// TIA Portal V17 export
// export: Created 2025-03-07T09:18:47.277747Z, ExportSetting WithDefaults, DisplayName Totally Integrated Automation Portal, DisplayVersion V17 Update 8, DisplayName TIA Portal Openness, DisplayVersion V17 Update 8, DisplayName TIA Portal Version Control Interface, DisplayVersion V17, DisplayName SINAMICS Startdrive Advanced, DisplayVersion V17 SP2, DisplayName SINAMICS Startdrive G110M, G120, G120C, G120D, G120P, G115D, DisplayVersion V17 SP2, DisplayName SINAMICS Startdrive G130, G150, S120, S150, SINAMICS MV, S210, DisplayVersion V17 SP2, DisplayName STEP 7 Professional, DisplayVersion V17 Update 8, DisplayName SINUMERIK ONE STEP 7 Toolbox, DisplayVersion V17 Update 12, DisplayName SINUMERIK 840D sl STEP 7 Toolbox, DisplayVersion V17 Update 12, DisplayName STEP 7 Safety, DisplayVersion V17 Update 6, DisplayName WinCC Advanced, DisplayVersion V17 Update 8
FUNCTION_BLOCK "FB6501_MEAS_DEVICE_HATCH"   // FB6501, LAD
{ S7_Optimized_Access := 'FALSE' }
AUTHOR : ETXETAR
VERSION : 1.0
// stored: AutoNumber false, IsIECCheckEnabled false, SetENOAutomatically false, UDAEnableTagReadback false
   VAR_INPUT
      OPTIONS_0 : Byte := 2#0000_0000;   // OPTIONS 0
      CLOSED_1_I : Bool;   // CLOSED 1 INPUT
      CLOSED_2_I : Bool;   // CLOSED 2 INPUT
      CLOSED_3_I : Bool;   // CLOSED 3 INPUT
      CLOSED_4_I : Bool;   // CLOSED 4 INPUT
      OPENED_1_I : Bool;   // OPEN 1 INPUT
      OPENED_2_I : Bool;   // OPEN 2 INPUT
      OPENED_3_I : Bool;   // OPEN 3 INPUT
      OPENED_4_I : Bool;   // OPEN 4 INPUT
      CLOSE_CONDITIONS : Bool;   // CLOSE CONDITIONS
      OPEN_CONDITIONS : Bool;   // OPEN CONDITIONS
      HMI_LINE_REQUEST : Bool;   // HMI LINE REQUEST
      CLOSE_AUTO_REQUEST : Bool;   // AUTO CLOSE REQUEST
      OPEN_AUTO_REQUEST_1 : Bool;   // AUTO OPEN REQUEST
      UNIT_ALARM : UInt;   // UNIT NUMBER MIN. NUMBER=1 MAX. NUMBER=4
      STATION_ALARM : UInt;   // STATION NUMBER MIN. NUMBER=0 MAX. NUMBER=4
   END_VAR
   VAR_OUTPUT
      CLOSED : Bool;   // CLOSED STATUS
      OPENED : Bool;   // OPENED STATUS
      CLOSED_1_ALARM : Bool;   // CLOSED 1 ALARM
      CLOSED_2_ALARM : Bool;   // CLOSED 2 ALARM
      CLOSED_3_ALARM : Bool;   // CLOSED 3 ALARM
      CLOSED_4_ALARM : Bool;   // CLOSED 4 ALARM
      OPENED_1_ALARM : Bool;   // OPENED 1 ALARM
      OPENED_2_ALARM : Bool;   // OPENED 2 ALARM
      OPENED_3_ALARM : Bool;   // OPENED 3 ALARM
      OPENED_4_ALARM : Bool;   // OPENED 4 ALARM
      HMI_MOTION_EXECUTABILITY_LEFT : Bool;   // HMI MOTION EXECUTABILITY LEFT
      HMI_MOTION_EXECUTABILITY_RIGHT : Bool;   // HMI MOTION EXECUTABILITY RIGHT
      HMI_MOTION_END_POS_LEFT : Bool;   // HMI MOTION END POSITION LEFT
      HMI_MOTION_END_POS_RIGHT : Bool;   // HMI MOTION END POSITION RIGHT
      HMI_MOTION_ACTIVE_LEFT : Bool;   // HMI MOTION ACTIVE LEFT
      HMI_MOTION_ACTIVE_RIGHT : Bool;   // HMI MOTION ACTIVE RIGHT
      CLOSE : Bool;   // CLOSE OUTPUT
      OPEN : Bool;   // OPEN OUTPUT
   END_VAR
   VAR DB_SPECIFIC
      CYL { S7_SetPoint := 'True'} : "OPEN_CLOSE_HATCH_CLADDING";
      TIMER_CLOSED { S7_SetPoint := 'True'} : TON_TIME;   // CLOSED TIMER
      TIMER_OPENED { S7_SetPoint := 'True'} : TON_TIME;   // OPENED TIMER
      TIMER_SIMULTANEITY { S7_SetPoint := 'True'} : TON_TIME;   // SIMULTANEITY TIMER
      TIMER_TIME_EXCEEDED { S7_SetPoint := 'True'} : TON_TIME;   // TIME EXCEEDED TIMER
   END_VAR
   VAR_TEMP
      INPUTS_MASK : Byte;   // INPUTS_MASK
      O_BYTE_0 : Struct   // OPTIONS BYTE 0
         CLOSED_INPUT_1 : Bool;   // CLOSED INPUT 1 OPTION
         CLOSED_INPUT_2 : Bool;   // CLOSED INPUT 2 OPTION
         CLOSED_INPUT_3 : Bool;   // CLOSED
         CLOSED_INPUT_4 : Bool;   // CLOSED INPUT 4 OPTION
         OPENED_INPUT_1 : Bool;   // OPENED INPUT 1 OPTION
         OPENED_INPUT_2 : Bool;   // OPENED INPUT 2 OPTION
         OPENED_INPUT_3 : Bool;   // OPENED INPUT 3 OPTION
         OPENED_INPUT_4 : Bool;   // OPENED INPUT 4 OPTION
      END_STRUCT;
      DB_NUMBER : DInt;   // DB NUMBER FOR ALARM AND HELP DECODING
   END_VAR
   // TIMER_CLOSED.PT := T#100MS;
   // TIMER_OPENED.PT := T#300MS;
   // TIMER_SIMULTANEITY.PT := T#100MS;
   // TIMER_TIME_EXCEEDED.PT := T#8S;
   VAR_TEMP   // added for the SCL form of the ladder/FBD networks
      _w1 : Bool;
      _w2 : Bool;
   END_VAR
BEGIN

NETWORK
TITLE = READ INSTANCE DB
      L     DINO;
      +     10#800000;
      T     #DB_NUMBER;


REGION Network 2: OPTIONS
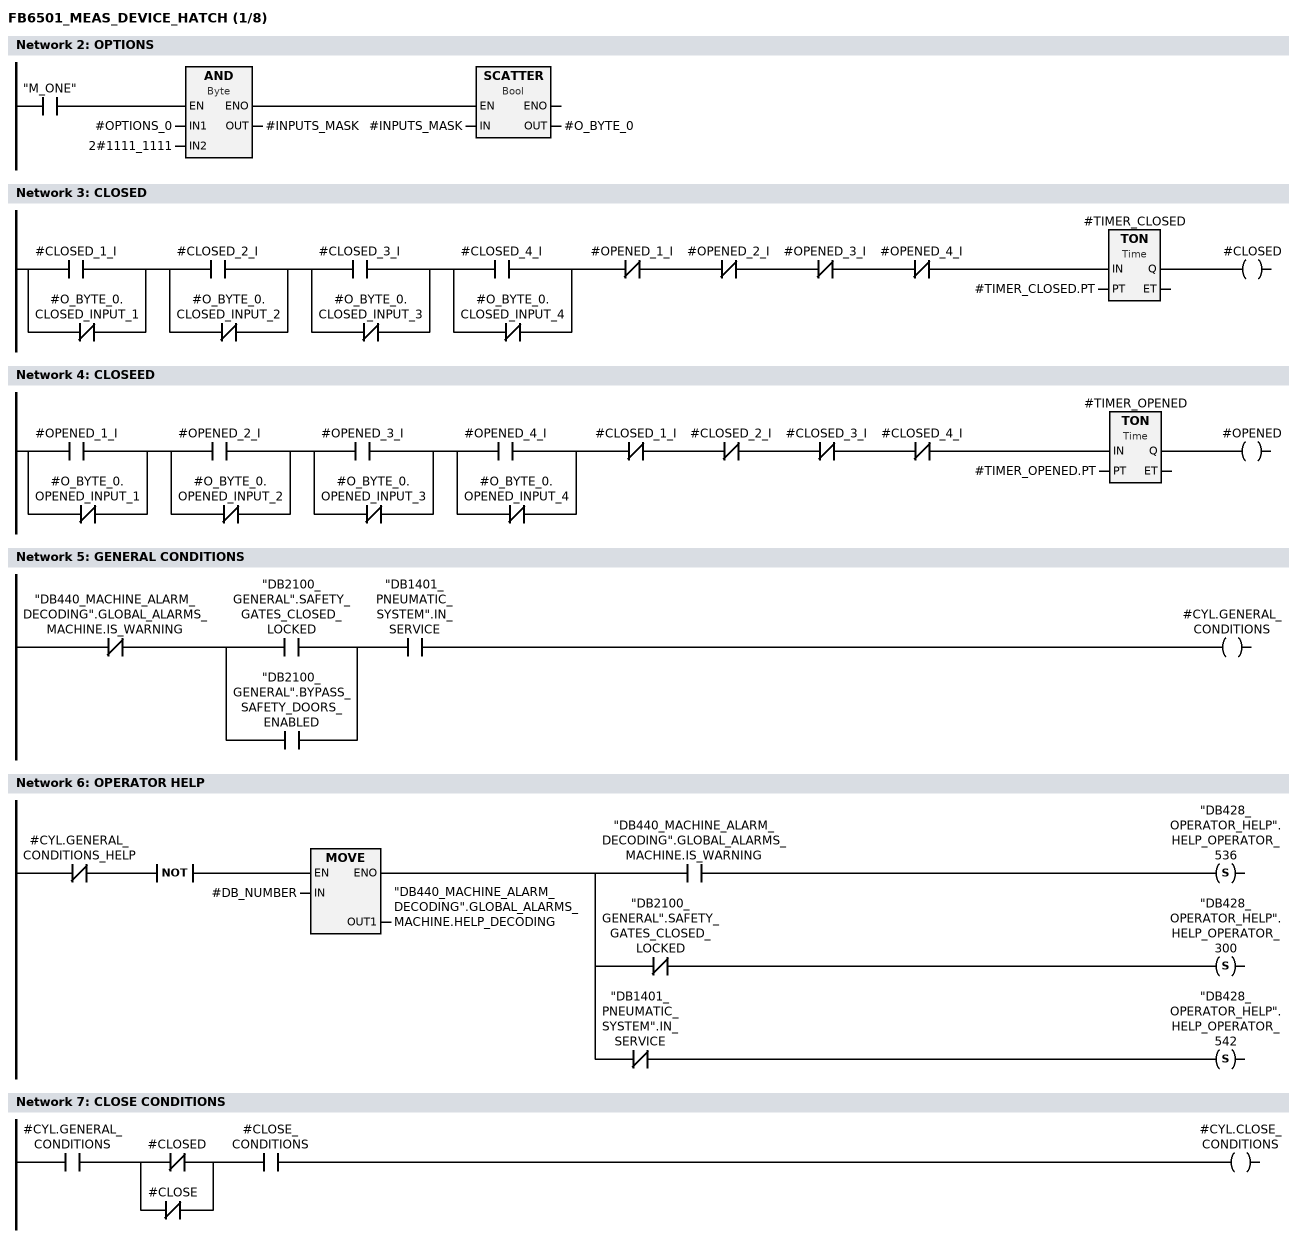
   RUNG wire#powerrail
      Contact( "M_ONE" )
      { S7_Templates := "SrcType := Byte"; S7_GenerateENO := "TRUE" } And(in1 := #OPTIONS_0, in2 := 2#1111_1111, out => #INPUTS_MASK)
      { S7_Templates := "[dest_type := Bool, src_type := Byte]" } SCATTER(IN := #INPUTS_MASK, OUT => #O_BYTE_0)
   END_RUNG
   // the same network as SCL:
   IF "M_ONE" THEN
       #INPUTS_MASK := #OPTIONS_0 AND 2#1111_1111;
       SCATTER(IN := #INPUTS_MASK, OUT => #O_BYTE_0);
   END_IF;
END_REGION

REGION Network 3: CLOSED
   RUNG wire#powerrail
      Contact( #CLOSED_1_I )
      wire#w1
      Contact( #CLOSED_2_I )
      wire#w2
      Contact( #CLOSED_3_I )
      wire#w3
      Contact( #CLOSED_4_I )
      wire#w4
      I_Contact( #OPENED_1_I )
      I_Contact( #OPENED_2_I )
      I_Contact( #OPENED_3_I )
      I_Contact( #OPENED_4_I )
      { S7_Templates := "time_type := Time" } #TIMER_CLOSED.TON(pt := #TIMER_CLOSED.PT, et =>)
      Coil( #CLOSED )
   END_RUNG
   RUNG wire#powerrail
      I_Contact( #O_BYTE_0.CLOSED_INPUT_1 )
   END_RUNG wire#w1
   RUNG wire#w1
      I_Contact( #O_BYTE_0.CLOSED_INPUT_2 )
   END_RUNG wire#w2
   RUNG wire#w2
      I_Contact( #O_BYTE_0.CLOSED_INPUT_3 )
   END_RUNG wire#w3
   RUNG wire#w3
      I_Contact( #O_BYTE_0.CLOSED_INPUT_4 )
   END_RUNG wire#w4
   // the same network as SCL:
   #TIMER_CLOSED(IN := (#CLOSED_1_I OR NOT #O_BYTE_0.CLOSED_INPUT_1) AND (#CLOSED_2_I OR NOT #O_BYTE_0.CLOSED_INPUT_2) AND (#CLOSED_3_I OR NOT #O_BYTE_0.CLOSED_INPUT_3) AND (#CLOSED_4_I OR NOT #O_BYTE_0.CLOSED_INPUT_4) AND NOT #OPENED_1_I AND NOT #OPENED_2_I AND NOT #OPENED_3_I AND NOT #OPENED_4_I,   // TON
                 PT := #TIMER_CLOSED.PT);
   #CLOSED := #TIMER_CLOSED.Q;
END_REGION

REGION Network 4: CLOSEED
   RUNG wire#powerrail
      Contact( #OPENED_1_I )
      wire#w1
      Contact( #OPENED_2_I )
      wire#w2
      Contact( #OPENED_3_I )
      wire#w3
      Contact( #OPENED_4_I )
      wire#w4
      I_Contact( #CLOSED_1_I )
      I_Contact( #CLOSED_2_I )
      I_Contact( #CLOSED_3_I )
      I_Contact( #CLOSED_4_I )
      { S7_Templates := "time_type := Time" } #TIMER_OPENED.TON(pt := #TIMER_OPENED.PT, et =>)
      Coil( #OPENED )
   END_RUNG
   RUNG wire#powerrail
      I_Contact( #O_BYTE_0.OPENED_INPUT_1 )
   END_RUNG wire#w1
   RUNG wire#w1
      I_Contact( #O_BYTE_0.OPENED_INPUT_2 )
   END_RUNG wire#w2
   RUNG wire#w2
      I_Contact( #O_BYTE_0.OPENED_INPUT_3 )
   END_RUNG wire#w3
   RUNG wire#w3
      I_Contact( #O_BYTE_0.OPENED_INPUT_4 )
   END_RUNG wire#w4
   // the same network as SCL:
   #TIMER_OPENED(IN := (#OPENED_1_I OR NOT #O_BYTE_0.OPENED_INPUT_1) AND (#OPENED_2_I OR NOT #O_BYTE_0.OPENED_INPUT_2) AND (#OPENED_3_I OR NOT #O_BYTE_0.OPENED_INPUT_3) AND (#OPENED_4_I OR NOT #O_BYTE_0.OPENED_INPUT_4) AND NOT #CLOSED_1_I AND NOT #CLOSED_2_I AND NOT #CLOSED_3_I AND NOT #CLOSED_4_I,   // TON
                 PT := #TIMER_OPENED.PT);
   #OPENED := #TIMER_OPENED.Q;
END_REGION

REGION Network 5: GENERAL CONDITIONS
   RUNG wire#powerrail
      I_Contact( "DB440_MACHINE_ALARM_DECODING".GLOBAL_ALARMS_MACHINE.IS_WARNING )
      wire#w1
      Contact( "DB2100_GENERAL".SAFETY_GATES_CLOSED_LOCKED )
      wire#w2
      Contact( "DB1401_PNEUMATIC_SYSTEM".IN_SERVICE )
      Coil( #CYL.GENERAL_CONDITIONS )
   END_RUNG
   RUNG wire#w1
      Contact( "DB2100_GENERAL".BYPASS_SAFETY_DOORS_ENABLED )
   END_RUNG wire#w2
   // the same network as SCL:
   #CYL.GENERAL_CONDITIONS := NOT "DB440_MACHINE_ALARM_DECODING".GLOBAL_ALARMS_MACHINE.IS_WARNING AND ("DB2100_GENERAL".SAFETY_GATES_CLOSED_LOCKED OR "DB2100_GENERAL".BYPASS_SAFETY_DOORS_ENABLED) AND "DB1401_PNEUMATIC_SYSTEM".IN_SERVICE;
END_REGION

REGION Network 6: OPERATOR HELP
   RUNG wire#powerrail
      I_Contact( #CYL.GENERAL_CONDITIONS_HELP )
      Not()
      { S7_GenerateENO := "TRUE" } Move(in := #DB_NUMBER, out1 => "DB440_MACHINE_ALARM_DECODING".GLOBAL_ALARMS_MACHINE.HELP_DECODING)
      wire#w1
      Contact( "DB440_MACHINE_ALARM_DECODING".GLOBAL_ALARMS_MACHINE.IS_WARNING )
      S_Coil( "DB428_OPERATOR_HELP".HELP_OPERATOR_536 )
   END_RUNG
   RUNG wire#w1
      I_Contact( "DB2100_GENERAL".SAFETY_GATES_CLOSED_LOCKED )
      S_Coil( "DB428_OPERATOR_HELP".HELP_OPERATOR_300 )
   END_RUNG
   RUNG wire#w1
      I_Contact( "DB1401_PNEUMATIC_SYSTEM".IN_SERVICE )
      S_Coil( "DB428_OPERATOR_HELP".HELP_OPERATOR_542 )
   END_RUNG
   // the same network as SCL:
   // ENO of a box is taken as its EN; it also drops when the box reports an error
   #_w1 := NOT (NOT #CYL.GENERAL_CONDITIONS_HELP);
   IF #_w1 THEN "DB440_MACHINE_ALARM_DECODING".GLOBAL_ALARMS_MACHINE.HELP_DECODING := #DB_NUMBER; END_IF;
   IF #_w1 AND "DB440_MACHINE_ALARM_DECODING".GLOBAL_ALARMS_MACHINE.IS_WARNING THEN
       "DB428_OPERATOR_HELP".HELP_OPERATOR_536 := TRUE;
   END_IF;
   IF #_w1 AND NOT "DB2100_GENERAL".SAFETY_GATES_CLOSED_LOCKED THEN
       "DB428_OPERATOR_HELP".HELP_OPERATOR_300 := TRUE;
   END_IF;
   IF #_w1 AND NOT "DB1401_PNEUMATIC_SYSTEM".IN_SERVICE THEN
       "DB428_OPERATOR_HELP".HELP_OPERATOR_542 := TRUE;
   END_IF;
END_REGION

REGION Network 7: CLOSE CONDITIONS
   RUNG wire#powerrail
      Contact( #CYL.GENERAL_CONDITIONS )
      wire#w1
      I_Contact( #CLOSED )
      wire#w2
      Contact( #CLOSE_CONDITIONS )
      Coil( #CYL.CLOSE_CONDITIONS )
   END_RUNG
   RUNG wire#w1
      I_Contact( #CLOSE )
   END_RUNG wire#w2
   // the same network as SCL:
   #CYL.CLOSE_CONDITIONS := #CYL.GENERAL_CONDITIONS AND (NOT #CLOSED OR NOT #CLOSE) AND #CLOSE_CONDITIONS;
END_REGION

REGION Network 8: OPERATOR HELP
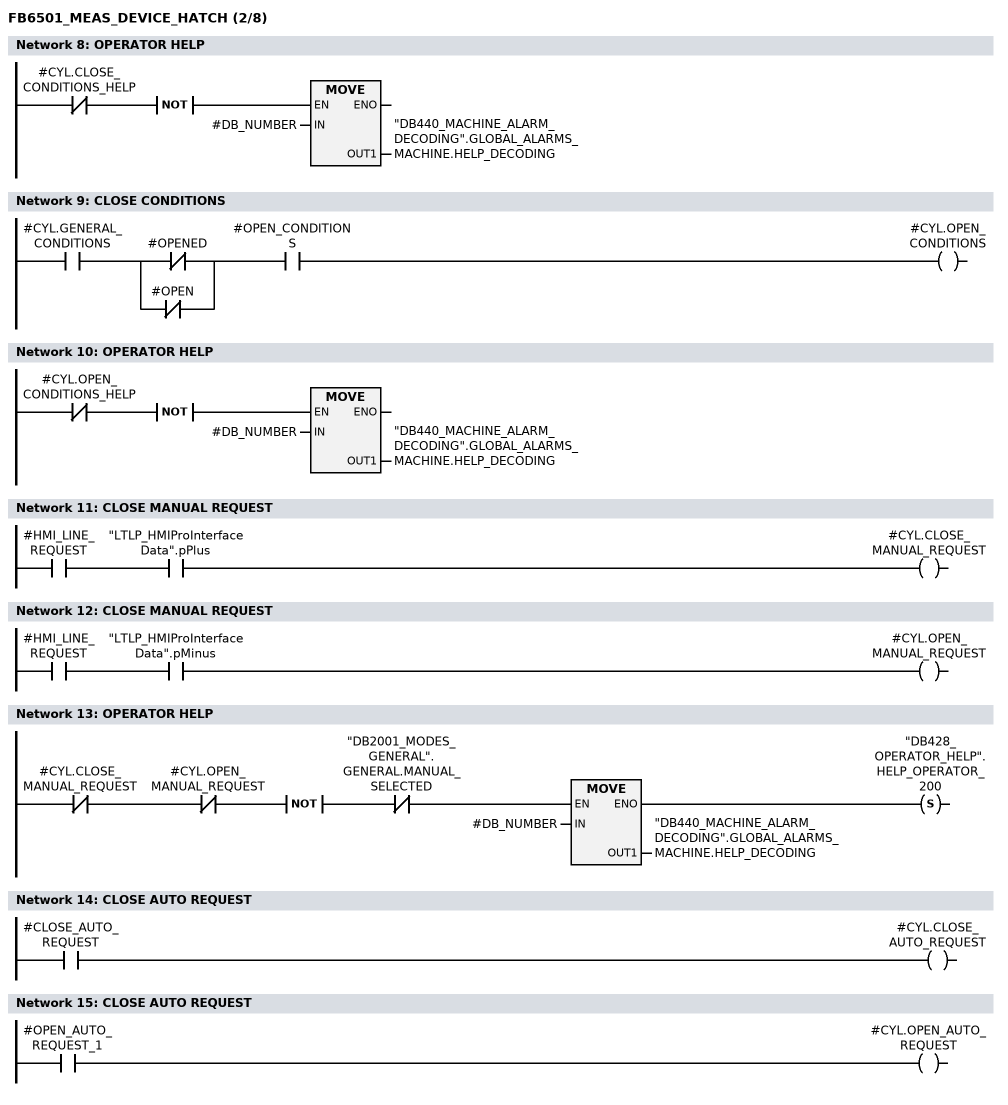
   RUNG wire#powerrail
      I_Contact( #CYL.CLOSE_CONDITIONS_HELP )
      Not()
      { S7_GenerateENO := "TRUE" } Move(in := #DB_NUMBER, out1 => "DB440_MACHINE_ALARM_DECODING".GLOBAL_ALARMS_MACHINE.HELP_DECODING)
   END_RUNG
   // the same network as SCL:
   IF NOT (NOT #CYL.CLOSE_CONDITIONS_HELP) THEN
       "DB440_MACHINE_ALARM_DECODING".GLOBAL_ALARMS_MACHINE.HELP_DECODING := #DB_NUMBER;
   END_IF;
END_REGION

REGION Network 9: CLOSE CONDITIONS
   RUNG wire#powerrail
      Contact( #CYL.GENERAL_CONDITIONS )
      wire#w1
      I_Contact( #OPENED )
      wire#w2
      Contact( #OPEN_CONDITIONS )
      Coil( #CYL.OPEN_CONDITIONS )
   END_RUNG
   RUNG wire#w1
      I_Contact( #OPEN )
   END_RUNG wire#w2
   // the same network as SCL:
   #CYL.OPEN_CONDITIONS := #CYL.GENERAL_CONDITIONS AND (NOT #OPENED OR NOT #OPEN) AND #OPEN_CONDITIONS;
END_REGION

REGION Network 10: OPERATOR HELP
   RUNG wire#powerrail
      I_Contact( #CYL.OPEN_CONDITIONS_HELP )
      Not()
      { S7_GenerateENO := "TRUE" } Move(in := #DB_NUMBER, out1 => "DB440_MACHINE_ALARM_DECODING".GLOBAL_ALARMS_MACHINE.HELP_DECODING)
   END_RUNG
   // the same network as SCL:
   IF NOT (NOT #CYL.OPEN_CONDITIONS_HELP) THEN
       "DB440_MACHINE_ALARM_DECODING".GLOBAL_ALARMS_MACHINE.HELP_DECODING := #DB_NUMBER;
   END_IF;
END_REGION

REGION Network 11: CLOSE MANUAL REQUEST
   RUNG wire#powerrail
      Contact( #HMI_LINE_REQUEST )
      Contact( "LTLP_HMIProInterfaceData".pPlus )
      Coil( #CYL.CLOSE_MANUAL_REQUEST )
   END_RUNG
   // the same network as SCL:
   #CYL.CLOSE_MANUAL_REQUEST := #HMI_LINE_REQUEST AND "LTLP_HMIProInterfaceData".pPlus;
END_REGION

REGION Network 12: CLOSE MANUAL REQUEST
   RUNG wire#powerrail
      Contact( #HMI_LINE_REQUEST )
      Contact( "LTLP_HMIProInterfaceData".pMinus )
      Coil( #CYL.OPEN_MANUAL_REQUEST )
   END_RUNG
   // the same network as SCL:
   #CYL.OPEN_MANUAL_REQUEST := #HMI_LINE_REQUEST AND "LTLP_HMIProInterfaceData".pMinus;
END_REGION

REGION Network 13: OPERATOR HELP
   RUNG wire#powerrail
      I_Contact( #CYL.CLOSE_MANUAL_REQUEST )
      I_Contact( #CYL.OPEN_MANUAL_REQUEST )
      Not()
      I_Contact( "DB2001_MODES_GENERAL".GENERAL.MANUAL_SELECTED )
      { S7_GenerateENO := "TRUE" } Move(in := #DB_NUMBER, out1 => "DB440_MACHINE_ALARM_DECODING".GLOBAL_ALARMS_MACHINE.HELP_DECODING)
      S_Coil( "DB428_OPERATOR_HELP".HELP_OPERATOR_200 )
   END_RUNG
   // the same network as SCL:
   // ENO of a box is taken as its EN; it also drops when the box reports an error
   IF NOT (NOT #CYL.CLOSE_MANUAL_REQUEST AND NOT #CYL.OPEN_MANUAL_REQUEST) AND NOT "DB2001_MODES_GENERAL".GENERAL.MANUAL_SELECTED THEN
       "DB440_MACHINE_ALARM_DECODING".GLOBAL_ALARMS_MACHINE.HELP_DECODING := #DB_NUMBER;
       "DB428_OPERATOR_HELP".HELP_OPERATOR_200 := TRUE;
   END_IF;
END_REGION

REGION Network 14: CLOSE AUTO REQUEST
   RUNG wire#powerrail
      Contact( #CLOSE_AUTO_REQUEST )
      Coil( #CYL.CLOSE_AUTO_REQUEST )
   END_RUNG
   // the same network as SCL:
   #CYL.CLOSE_AUTO_REQUEST := #CLOSE_AUTO_REQUEST;
END_REGION

REGION Network 15: CLOSE AUTO REQUEST
   RUNG wire#powerrail
      Contact( #OPEN_AUTO_REQUEST_1 )
      Coil( #CYL.OPEN_AUTO_REQUEST )
   END_RUNG
   // the same network as SCL:
   #CYL.OPEN_AUTO_REQUEST := #OPEN_AUTO_REQUEST_1;
END_REGION

REGION Network 16: CLOSE GLOBAL REQUEST
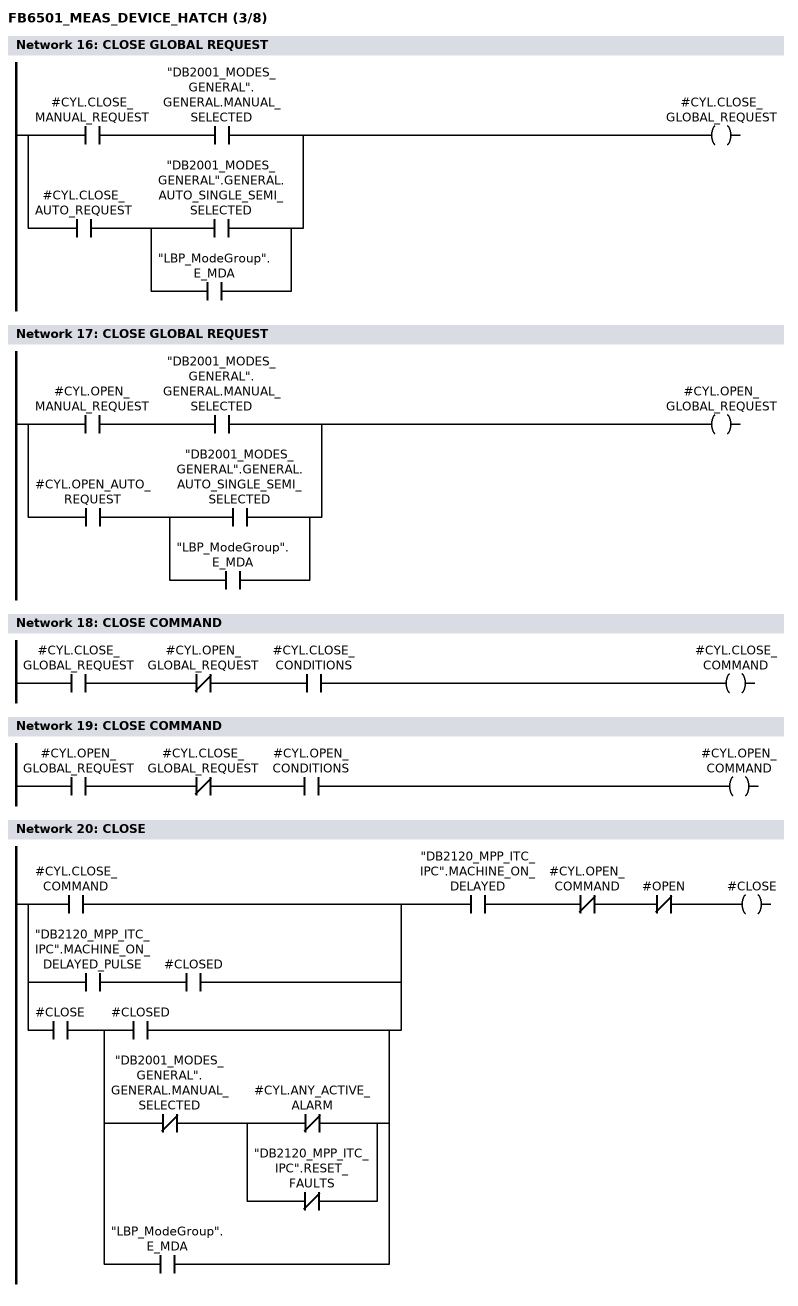
   RUNG wire#powerrail
      Contact( #CYL.CLOSE_MANUAL_REQUEST )
      Contact( "DB2001_MODES_GENERAL".GENERAL.MANUAL_SELECTED )
      wire#w1
      Coil( #CYL.CLOSE_GLOBAL_REQUEST )
   END_RUNG
   RUNG wire#powerrail
      Contact( #CYL.CLOSE_AUTO_REQUEST )
      wire#w2
      Contact( "DB2001_MODES_GENERAL".GENERAL.AUTO_SINGLE_SEMI_SELECTED )
   END_RUNG wire#w1
   RUNG wire#w2
      Contact( "LBP_ModeGroup".E_MDA )
   END_RUNG wire#w1
   // the same network as SCL:
   #CYL.CLOSE_GLOBAL_REQUEST := (#CYL.CLOSE_MANUAL_REQUEST AND "DB2001_MODES_GENERAL".GENERAL.MANUAL_SELECTED) OR (#CYL.CLOSE_AUTO_REQUEST AND ("DB2001_MODES_GENERAL".GENERAL.AUTO_SINGLE_SEMI_SELECTED OR "LBP_ModeGroup".E_MDA));
END_REGION

REGION Network 17: CLOSE GLOBAL REQUEST
   RUNG wire#powerrail
      Contact( #CYL.OPEN_MANUAL_REQUEST )
      Contact( "DB2001_MODES_GENERAL".GENERAL.MANUAL_SELECTED )
      wire#w1
      Coil( #CYL.OPEN_GLOBAL_REQUEST )
   END_RUNG
   RUNG wire#powerrail
      Contact( #CYL.OPEN_AUTO_REQUEST )
      wire#w2
      Contact( "DB2001_MODES_GENERAL".GENERAL.AUTO_SINGLE_SEMI_SELECTED )
   END_RUNG wire#w1
   RUNG wire#w2
      Contact( "LBP_ModeGroup".E_MDA )
   END_RUNG wire#w1
   // the same network as SCL:
   #CYL.OPEN_GLOBAL_REQUEST := (#CYL.OPEN_MANUAL_REQUEST AND "DB2001_MODES_GENERAL".GENERAL.MANUAL_SELECTED) OR (#CYL.OPEN_AUTO_REQUEST AND ("DB2001_MODES_GENERAL".GENERAL.AUTO_SINGLE_SEMI_SELECTED OR "LBP_ModeGroup".E_MDA));
END_REGION

REGION Network 18: CLOSE COMMAND
   RUNG wire#powerrail
      Contact( #CYL.CLOSE_GLOBAL_REQUEST )
      I_Contact( #CYL.OPEN_GLOBAL_REQUEST )
      Contact( #CYL.CLOSE_CONDITIONS )
      Coil( #CYL.CLOSE_COMMAND )
   END_RUNG
   // the same network as SCL:
   #CYL.CLOSE_COMMAND := #CYL.CLOSE_GLOBAL_REQUEST AND NOT #CYL.OPEN_GLOBAL_REQUEST AND #CYL.CLOSE_CONDITIONS;
END_REGION

REGION Network 19: CLOSE COMMAND
   RUNG wire#powerrail
      Contact( #CYL.OPEN_GLOBAL_REQUEST )
      I_Contact( #CYL.CLOSE_GLOBAL_REQUEST )
      Contact( #CYL.OPEN_CONDITIONS )
      Coil( #CYL.OPEN_COMMAND )
   END_RUNG
   // the same network as SCL:
   #CYL.OPEN_COMMAND := #CYL.OPEN_GLOBAL_REQUEST AND NOT #CYL.CLOSE_GLOBAL_REQUEST AND #CYL.OPEN_CONDITIONS;
END_REGION

REGION Network 20: CLOSE
   RUNG wire#powerrail
      Contact( #CYL.CLOSE_COMMAND )
      wire#w1
      Contact( "DB2120_MPP_ITC_IPC".MACHINE_ON_DELAYED )
      I_Contact( #CYL.OPEN_COMMAND )
      I_Contact( #OPEN )
      Coil( #CLOSE )
   END_RUNG
   RUNG wire#powerrail
      Contact( "DB2120_MPP_ITC_IPC".MACHINE_ON_DELAYED_PULSE )
      Contact( #CLOSED )
   END_RUNG wire#w1
   RUNG wire#powerrail
      Contact( #CLOSE )
      wire#w2
      Contact( #CLOSED )
   END_RUNG wire#w1
   RUNG wire#w2
      I_Contact( "DB2001_MODES_GENERAL".GENERAL.MANUAL_SELECTED )
      wire#w3
      I_Contact( #CYL.ANY_ACTIVE_ALARM )
   END_RUNG wire#w1
   RUNG wire#w3
      I_Contact( "DB2120_MPP_ITC_IPC".RESET_FAULTS )
   END_RUNG wire#w1
   RUNG wire#w2
      Contact( "LBP_ModeGroup".E_MDA )
   END_RUNG wire#w1
   // the same network as SCL:
   #CLOSE := (#CYL.CLOSE_COMMAND OR ("DB2120_MPP_ITC_IPC".MACHINE_ON_DELAYED_PULSE AND #CLOSED) OR (#CLOSE AND (#CLOSED OR (NOT "DB2001_MODES_GENERAL".GENERAL.MANUAL_SELECTED AND (NOT #CYL.ANY_ACTIVE_ALARM OR NOT "DB2120_MPP_ITC_IPC".RESET_FAULTS)) OR "LBP_ModeGroup".E_MDA))) AND "DB2120_MPP_ITC_IPC".MACHINE_ON_DELAYED AND NOT #CYL.OPEN_COMMAND AND NOT #OPEN;
END_REGION

REGION Network 21: CLOSE
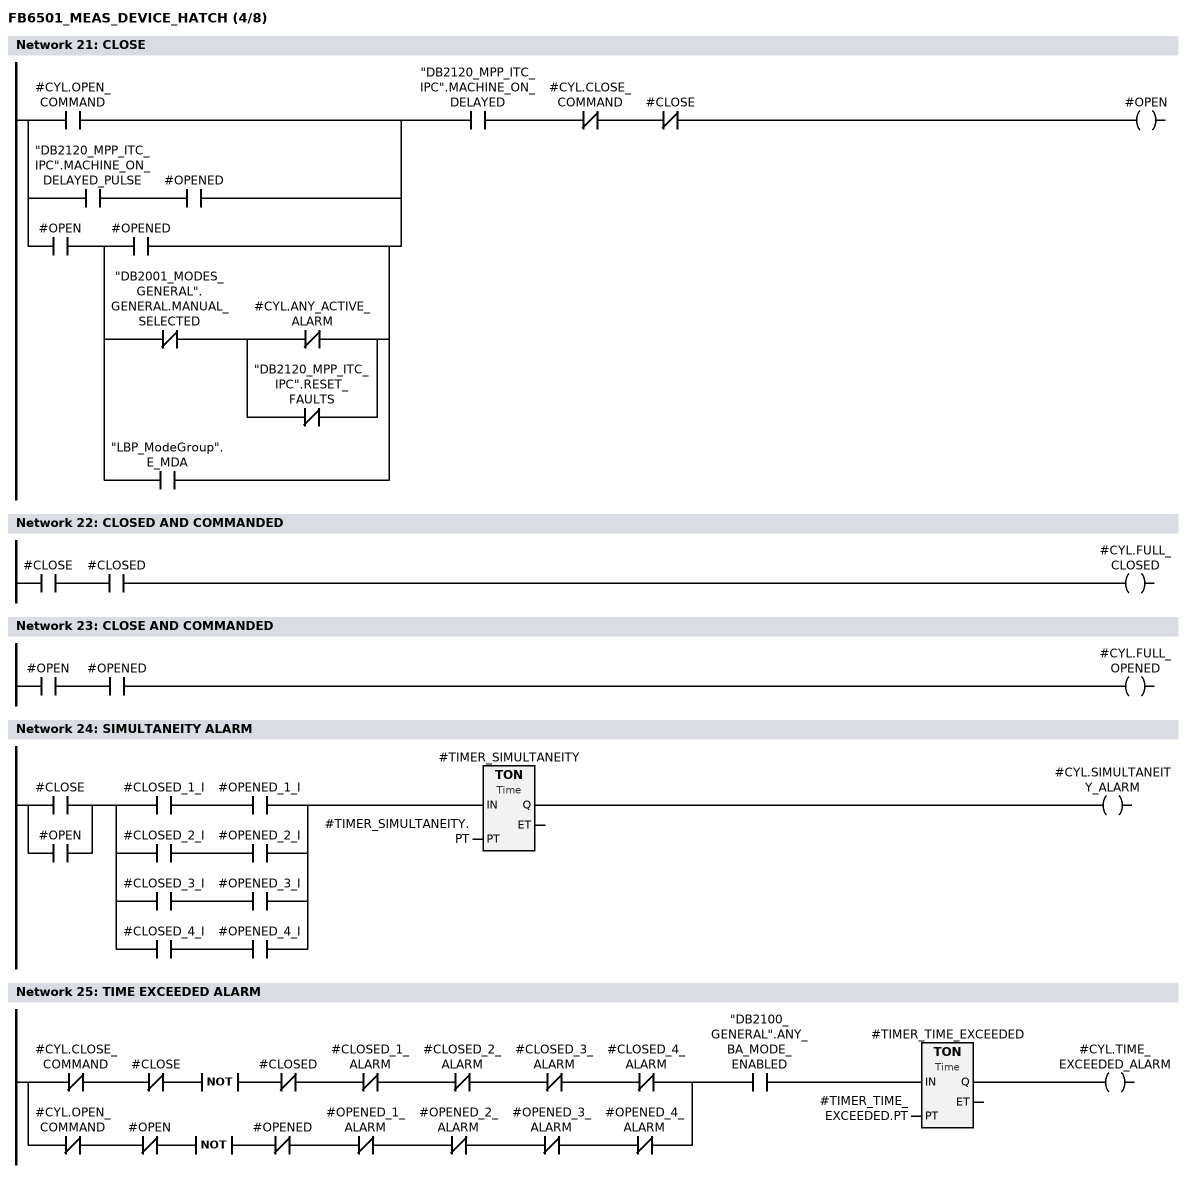
   RUNG wire#powerrail
      Contact( #CYL.OPEN_COMMAND )
      wire#w1
      Contact( "DB2120_MPP_ITC_IPC".MACHINE_ON_DELAYED )
      I_Contact( #CYL.CLOSE_COMMAND )
      I_Contact( #CLOSE )
      Coil( #OPEN )
   END_RUNG
   RUNG wire#powerrail
      Contact( "DB2120_MPP_ITC_IPC".MACHINE_ON_DELAYED_PULSE )
      Contact( #OPENED )
   END_RUNG wire#w1
   RUNG wire#powerrail
      Contact( #OPEN )
      wire#w2
      Contact( #OPENED )
   END_RUNG wire#w1
   RUNG wire#w2
      I_Contact( "DB2001_MODES_GENERAL".GENERAL.MANUAL_SELECTED )
      wire#w3
      I_Contact( #CYL.ANY_ACTIVE_ALARM )
   END_RUNG wire#w1
   RUNG wire#w3
      I_Contact( "DB2120_MPP_ITC_IPC".RESET_FAULTS )
   END_RUNG wire#w1
   RUNG wire#w2
      Contact( "LBP_ModeGroup".E_MDA )
   END_RUNG wire#w1
   // the same network as SCL:
   #OPEN := (#CYL.OPEN_COMMAND OR ("DB2120_MPP_ITC_IPC".MACHINE_ON_DELAYED_PULSE AND #OPENED) OR (#OPEN AND (#OPENED OR (NOT "DB2001_MODES_GENERAL".GENERAL.MANUAL_SELECTED AND (NOT #CYL.ANY_ACTIVE_ALARM OR NOT "DB2120_MPP_ITC_IPC".RESET_FAULTS)) OR "LBP_ModeGroup".E_MDA))) AND "DB2120_MPP_ITC_IPC".MACHINE_ON_DELAYED AND NOT #CYL.CLOSE_COMMAND AND NOT #CLOSE;
END_REGION

REGION Network 22: CLOSED AND COMMANDED
   RUNG wire#powerrail
      Contact( #CLOSE )
      Contact( #CLOSED )
      Coil( #CYL.FULL_CLOSED )
   END_RUNG
   // the same network as SCL:
   #CYL.FULL_CLOSED := #CLOSE AND #CLOSED;
END_REGION

REGION Network 23: CLOSE AND COMMANDED
   RUNG wire#powerrail
      Contact( #OPEN )
      Contact( #OPENED )
      Coil( #CYL.FULL_OPENED )
   END_RUNG
   // the same network as SCL:
   #CYL.FULL_OPENED := #OPEN AND #OPENED;
END_REGION

REGION Network 24: SIMULTANEITY ALARM
   RUNG wire#powerrail
      Contact( #CLOSE )
      wire#w1
      Contact( #CLOSED_1_I )
      Contact( #OPENED_1_I )
      wire#w2
      { S7_Templates := "time_type := Time" } #TIMER_SIMULTANEITY.TON(pt := #TIMER_SIMULTANEITY.PT, et =>)
      Coil( #CYL.SIMULTANEITY_ALARM )
   END_RUNG
   RUNG wire#powerrail
      Contact( #OPEN )
   END_RUNG wire#w1
   RUNG wire#w1
      Contact( #CLOSED_2_I )
      Contact( #OPENED_2_I )
   END_RUNG wire#w2
   RUNG wire#w1
      Contact( #CLOSED_3_I )
      Contact( #OPENED_3_I )
   END_RUNG wire#w2
   RUNG wire#w1
      Contact( #CLOSED_4_I )
      Contact( #OPENED_4_I )
   END_RUNG wire#w2
   // the same network as SCL:
   #TIMER_SIMULTANEITY(IN := (#CLOSE OR #OPEN) AND ((#CLOSED_1_I AND #OPENED_1_I) OR (#CLOSED_2_I AND #OPENED_2_I) OR (#CLOSED_3_I AND #OPENED_3_I) OR (#CLOSED_4_I AND #OPENED_4_I)),   // TON
                       PT := #TIMER_SIMULTANEITY.PT);
   #CYL.SIMULTANEITY_ALARM := #TIMER_SIMULTANEITY.Q;
END_REGION

REGION Network 25: TIME EXCEEDED ALARM
   RUNG wire#powerrail
      I_Contact( #CYL.CLOSE_COMMAND )
      I_Contact( #CLOSE )
      Not()
      I_Contact( #CLOSED )
      I_Contact( #CLOSED_1_ALARM )
      I_Contact( #CLOSED_2_ALARM )
      I_Contact( #CLOSED_3_ALARM )
      I_Contact( #CLOSED_4_ALARM )
      wire#w1
      Contact( "DB2100_GENERAL".ANY_BA_MODE_ENABLED )
      { S7_Templates := "time_type := Time" } #TIMER_TIME_EXCEEDED.TON(pt := #TIMER_TIME_EXCEEDED.PT, et =>)
      Coil( #CYL.TIME_EXCEEDED_ALARM )
   END_RUNG
   RUNG wire#powerrail
      I_Contact( #CYL.OPEN_COMMAND )
      I_Contact( #OPEN )
      Not()
      I_Contact( #OPENED )
      I_Contact( #OPENED_1_ALARM )
      I_Contact( #OPENED_2_ALARM )
      I_Contact( #OPENED_3_ALARM )
      I_Contact( #OPENED_4_ALARM )
   END_RUNG wire#w1
   // the same network as SCL:
   #TIMER_TIME_EXCEEDED(IN := ((NOT (NOT #CYL.CLOSE_COMMAND AND NOT #CLOSE) AND NOT #CLOSED AND NOT #CLOSED_1_ALARM AND NOT #CLOSED_2_ALARM AND NOT #CLOSED_3_ALARM AND NOT #CLOSED_4_ALARM) OR (NOT (NOT #CYL.OPEN_COMMAND AND NOT #OPEN) AND NOT #OPENED AND NOT #OPENED_1_ALARM AND NOT #OPENED_2_ALARM AND NOT #OPENED_3_ALARM AND NOT #OPENED_4_ALARM)) AND "DB2100_GENERAL".ANY_BA_MODE_ENABLED,   // TON
                        PT := #TIMER_TIME_EXCEEDED.PT);
   #CYL.TIME_EXCEEDED_ALARM := #TIMER_TIME_EXCEEDED.Q;
END_REGION

REGION Network 26: CLOSED 1 ALARM
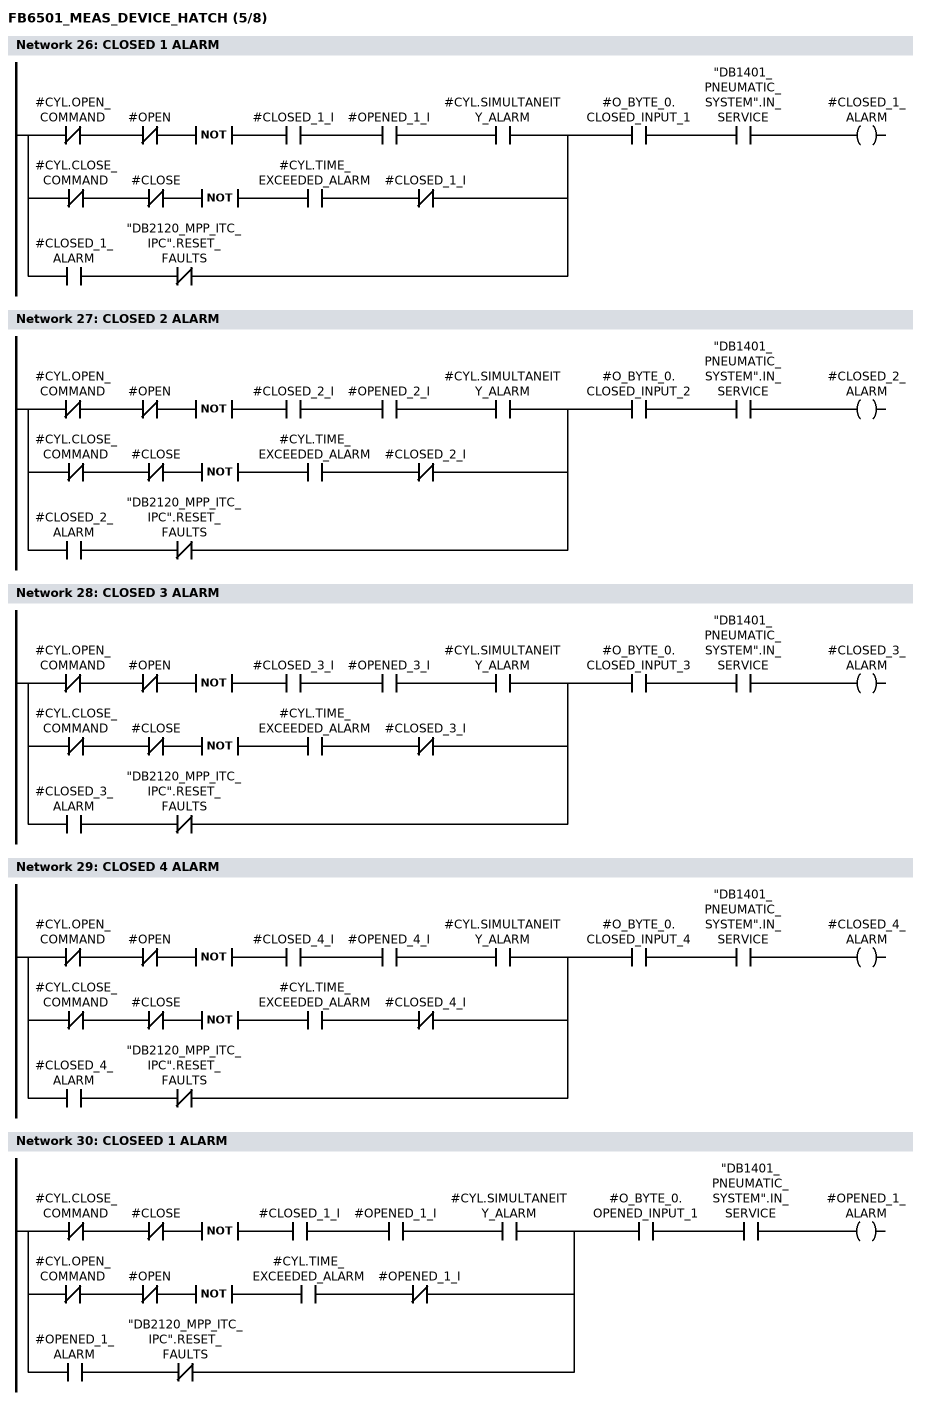
   RUNG wire#powerrail
      I_Contact( #CYL.OPEN_COMMAND )
      I_Contact( #OPEN )
      Not()
      Contact( #CLOSED_1_I )
      Contact( #OPENED_1_I )
      Contact( #CYL.SIMULTANEITY_ALARM )
      wire#w1
      Contact( #O_BYTE_0.CLOSED_INPUT_1 )
      Contact( "DB1401_PNEUMATIC_SYSTEM".IN_SERVICE )
      Coil( #CLOSED_1_ALARM )
   END_RUNG
   RUNG wire#powerrail
      I_Contact( #CYL.CLOSE_COMMAND )
      I_Contact( #CLOSE )
      Not()
      Contact( #CYL.TIME_EXCEEDED_ALARM )
      I_Contact( #CLOSED_1_I )
   END_RUNG wire#w1
   RUNG wire#powerrail
      Contact( #CLOSED_1_ALARM )
      I_Contact( "DB2120_MPP_ITC_IPC".RESET_FAULTS )
   END_RUNG wire#w1
   // the same network as SCL:
   #CLOSED_1_ALARM := ((NOT (NOT #CYL.OPEN_COMMAND AND NOT #OPEN) AND #CLOSED_1_I AND #OPENED_1_I AND #CYL.SIMULTANEITY_ALARM) OR (NOT (NOT #CYL.CLOSE_COMMAND AND NOT #CLOSE) AND #CYL.TIME_EXCEEDED_ALARM AND NOT #CLOSED_1_I) OR (#CLOSED_1_ALARM AND NOT "DB2120_MPP_ITC_IPC".RESET_FAULTS)) AND #O_BYTE_0.CLOSED_INPUT_1 AND "DB1401_PNEUMATIC_SYSTEM".IN_SERVICE;
END_REGION

REGION Network 27: CLOSED 2 ALARM
   RUNG wire#powerrail
      I_Contact( #CYL.OPEN_COMMAND )
      I_Contact( #OPEN )
      Not()
      Contact( #CLOSED_2_I )
      Contact( #OPENED_2_I )
      Contact( #CYL.SIMULTANEITY_ALARM )
      wire#w1
      Contact( #O_BYTE_0.CLOSED_INPUT_2 )
      Contact( "DB1401_PNEUMATIC_SYSTEM".IN_SERVICE )
      Coil( #CLOSED_2_ALARM )
   END_RUNG
   RUNG wire#powerrail
      I_Contact( #CYL.CLOSE_COMMAND )
      I_Contact( #CLOSE )
      Not()
      Contact( #CYL.TIME_EXCEEDED_ALARM )
      I_Contact( #CLOSED_2_I )
   END_RUNG wire#w1
   RUNG wire#powerrail
      Contact( #CLOSED_2_ALARM )
      I_Contact( "DB2120_MPP_ITC_IPC".RESET_FAULTS )
   END_RUNG wire#w1
   // the same network as SCL:
   #CLOSED_2_ALARM := ((NOT (NOT #CYL.OPEN_COMMAND AND NOT #OPEN) AND #CLOSED_2_I AND #OPENED_2_I AND #CYL.SIMULTANEITY_ALARM) OR (NOT (NOT #CYL.CLOSE_COMMAND AND NOT #CLOSE) AND #CYL.TIME_EXCEEDED_ALARM AND NOT #CLOSED_2_I) OR (#CLOSED_2_ALARM AND NOT "DB2120_MPP_ITC_IPC".RESET_FAULTS)) AND #O_BYTE_0.CLOSED_INPUT_2 AND "DB1401_PNEUMATIC_SYSTEM".IN_SERVICE;
END_REGION

REGION Network 28: CLOSED 3 ALARM
   RUNG wire#powerrail
      I_Contact( #CYL.OPEN_COMMAND )
      I_Contact( #OPEN )
      Not()
      Contact( #CLOSED_3_I )
      Contact( #OPENED_3_I )
      Contact( #CYL.SIMULTANEITY_ALARM )
      wire#w1
      Contact( #O_BYTE_0.CLOSED_INPUT_3 )
      Contact( "DB1401_PNEUMATIC_SYSTEM".IN_SERVICE )
      Coil( #CLOSED_3_ALARM )
   END_RUNG
   RUNG wire#powerrail
      I_Contact( #CYL.CLOSE_COMMAND )
      I_Contact( #CLOSE )
      Not()
      Contact( #CYL.TIME_EXCEEDED_ALARM )
      I_Contact( #CLOSED_3_I )
   END_RUNG wire#w1
   RUNG wire#powerrail
      Contact( #CLOSED_3_ALARM )
      I_Contact( "DB2120_MPP_ITC_IPC".RESET_FAULTS )
   END_RUNG wire#w1
   // the same network as SCL:
   #CLOSED_3_ALARM := ((NOT (NOT #CYL.OPEN_COMMAND AND NOT #OPEN) AND #CLOSED_3_I AND #OPENED_3_I AND #CYL.SIMULTANEITY_ALARM) OR (NOT (NOT #CYL.CLOSE_COMMAND AND NOT #CLOSE) AND #CYL.TIME_EXCEEDED_ALARM AND NOT #CLOSED_3_I) OR (#CLOSED_3_ALARM AND NOT "DB2120_MPP_ITC_IPC".RESET_FAULTS)) AND #O_BYTE_0.CLOSED_INPUT_3 AND "DB1401_PNEUMATIC_SYSTEM".IN_SERVICE;
END_REGION

REGION Network 29: CLOSED 4 ALARM
   RUNG wire#powerrail
      I_Contact( #CYL.OPEN_COMMAND )
      I_Contact( #OPEN )
      Not()
      Contact( #CLOSED_4_I )
      Contact( #OPENED_4_I )
      Contact( #CYL.SIMULTANEITY_ALARM )
      wire#w1
      Contact( #O_BYTE_0.CLOSED_INPUT_4 )
      Contact( "DB1401_PNEUMATIC_SYSTEM".IN_SERVICE )
      Coil( #CLOSED_4_ALARM )
   END_RUNG
   RUNG wire#powerrail
      I_Contact( #CYL.CLOSE_COMMAND )
      I_Contact( #CLOSE )
      Not()
      Contact( #CYL.TIME_EXCEEDED_ALARM )
      I_Contact( #CLOSED_4_I )
   END_RUNG wire#w1
   RUNG wire#powerrail
      Contact( #CLOSED_4_ALARM )
      I_Contact( "DB2120_MPP_ITC_IPC".RESET_FAULTS )
   END_RUNG wire#w1
   // the same network as SCL:
   #CLOSED_4_ALARM := ((NOT (NOT #CYL.OPEN_COMMAND AND NOT #OPEN) AND #CLOSED_4_I AND #OPENED_4_I AND #CYL.SIMULTANEITY_ALARM) OR (NOT (NOT #CYL.CLOSE_COMMAND AND NOT #CLOSE) AND #CYL.TIME_EXCEEDED_ALARM AND NOT #CLOSED_4_I) OR (#CLOSED_4_ALARM AND NOT "DB2120_MPP_ITC_IPC".RESET_FAULTS)) AND #O_BYTE_0.CLOSED_INPUT_4 AND "DB1401_PNEUMATIC_SYSTEM".IN_SERVICE;
END_REGION

REGION Network 30: CLOSEED 1 ALARM
   RUNG wire#powerrail
      I_Contact( #CYL.CLOSE_COMMAND )
      I_Contact( #CLOSE )
      Not()
      Contact( #CLOSED_1_I )
      Contact( #OPENED_1_I )
      Contact( #CYL.SIMULTANEITY_ALARM )
      wire#w1
      Contact( #O_BYTE_0.OPENED_INPUT_1 )
      Contact( "DB1401_PNEUMATIC_SYSTEM".IN_SERVICE )
      Coil( #OPENED_1_ALARM )
   END_RUNG
   RUNG wire#powerrail
      I_Contact( #CYL.OPEN_COMMAND )
      I_Contact( #OPEN )
      Not()
      Contact( #CYL.TIME_EXCEEDED_ALARM )
      I_Contact( #OPENED_1_I )
   END_RUNG wire#w1
   RUNG wire#powerrail
      Contact( #OPENED_1_ALARM )
      I_Contact( "DB2120_MPP_ITC_IPC".RESET_FAULTS )
   END_RUNG wire#w1
   // the same network as SCL:
   #OPENED_1_ALARM := ((NOT (NOT #CYL.CLOSE_COMMAND AND NOT #CLOSE) AND #CLOSED_1_I AND #OPENED_1_I AND #CYL.SIMULTANEITY_ALARM) OR (NOT (NOT #CYL.OPEN_COMMAND AND NOT #OPEN) AND #CYL.TIME_EXCEEDED_ALARM AND NOT #OPENED_1_I) OR (#OPENED_1_ALARM AND NOT "DB2120_MPP_ITC_IPC".RESET_FAULTS)) AND #O_BYTE_0.OPENED_INPUT_1 AND "DB1401_PNEUMATIC_SYSTEM".IN_SERVICE;
END_REGION

REGION Network 31: CLOSEED 2 ALARM
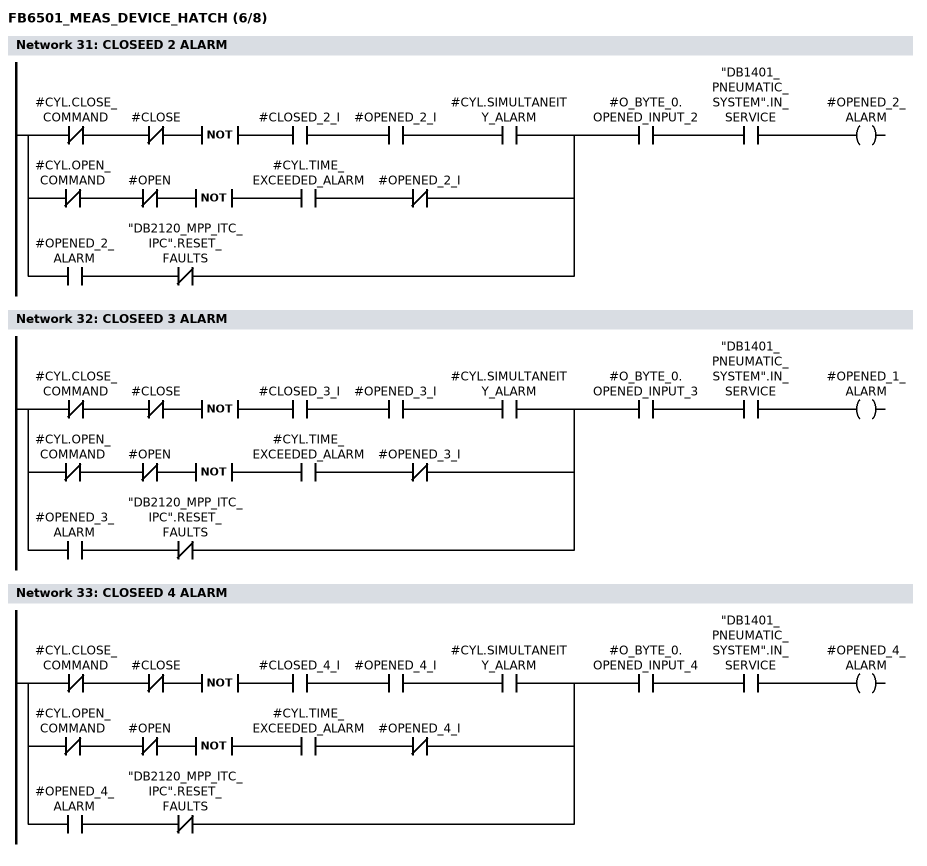
   RUNG wire#powerrail
      I_Contact( #CYL.CLOSE_COMMAND )
      I_Contact( #CLOSE )
      Not()
      Contact( #CLOSED_2_I )
      Contact( #OPENED_2_I )
      Contact( #CYL.SIMULTANEITY_ALARM )
      wire#w1
      Contact( #O_BYTE_0.OPENED_INPUT_2 )
      Contact( "DB1401_PNEUMATIC_SYSTEM".IN_SERVICE )
      Coil( #OPENED_2_ALARM )
   END_RUNG
   RUNG wire#powerrail
      I_Contact( #CYL.OPEN_COMMAND )
      I_Contact( #OPEN )
      Not()
      Contact( #CYL.TIME_EXCEEDED_ALARM )
      I_Contact( #OPENED_2_I )
   END_RUNG wire#w1
   RUNG wire#powerrail
      Contact( #OPENED_2_ALARM )
      I_Contact( "DB2120_MPP_ITC_IPC".RESET_FAULTS )
   END_RUNG wire#w1
   // the same network as SCL:
   #OPENED_2_ALARM := ((NOT (NOT #CYL.CLOSE_COMMAND AND NOT #CLOSE) AND #CLOSED_2_I AND #OPENED_2_I AND #CYL.SIMULTANEITY_ALARM) OR (NOT (NOT #CYL.OPEN_COMMAND AND NOT #OPEN) AND #CYL.TIME_EXCEEDED_ALARM AND NOT #OPENED_2_I) OR (#OPENED_2_ALARM AND NOT "DB2120_MPP_ITC_IPC".RESET_FAULTS)) AND #O_BYTE_0.OPENED_INPUT_2 AND "DB1401_PNEUMATIC_SYSTEM".IN_SERVICE;
END_REGION

REGION Network 32: CLOSEED 3 ALARM
   RUNG wire#powerrail
      I_Contact( #CYL.CLOSE_COMMAND )
      I_Contact( #CLOSE )
      Not()
      Contact( #CLOSED_3_I )
      Contact( #OPENED_3_I )
      Contact( #CYL.SIMULTANEITY_ALARM )
      wire#w1
      Contact( #O_BYTE_0.OPENED_INPUT_3 )
      Contact( "DB1401_PNEUMATIC_SYSTEM".IN_SERVICE )
      Coil( #OPENED_1_ALARM )
   END_RUNG
   RUNG wire#powerrail
      I_Contact( #CYL.OPEN_COMMAND )
      I_Contact( #OPEN )
      Not()
      Contact( #CYL.TIME_EXCEEDED_ALARM )
      I_Contact( #OPENED_3_I )
   END_RUNG wire#w1
   RUNG wire#powerrail
      Contact( #OPENED_3_ALARM )
      I_Contact( "DB2120_MPP_ITC_IPC".RESET_FAULTS )
   END_RUNG wire#w1
   // the same network as SCL:
   #OPENED_1_ALARM := ((NOT (NOT #CYL.CLOSE_COMMAND AND NOT #CLOSE) AND #CLOSED_3_I AND #OPENED_3_I AND #CYL.SIMULTANEITY_ALARM) OR (NOT (NOT #CYL.OPEN_COMMAND AND NOT #OPEN) AND #CYL.TIME_EXCEEDED_ALARM AND NOT #OPENED_3_I) OR (#OPENED_3_ALARM AND NOT "DB2120_MPP_ITC_IPC".RESET_FAULTS)) AND #O_BYTE_0.OPENED_INPUT_3 AND "DB1401_PNEUMATIC_SYSTEM".IN_SERVICE;
END_REGION

REGION Network 33: CLOSEED 4 ALARM
   RUNG wire#powerrail
      I_Contact( #CYL.CLOSE_COMMAND )
      I_Contact( #CLOSE )
      Not()
      Contact( #CLOSED_4_I )
      Contact( #OPENED_4_I )
      Contact( #CYL.SIMULTANEITY_ALARM )
      wire#w1
      Contact( #O_BYTE_0.OPENED_INPUT_4 )
      Contact( "DB1401_PNEUMATIC_SYSTEM".IN_SERVICE )
      Coil( #OPENED_4_ALARM )
   END_RUNG
   RUNG wire#powerrail
      I_Contact( #CYL.OPEN_COMMAND )
      I_Contact( #OPEN )
      Not()
      Contact( #CYL.TIME_EXCEEDED_ALARM )
      I_Contact( #OPENED_4_I )
   END_RUNG wire#w1
   RUNG wire#powerrail
      Contact( #OPENED_4_ALARM )
      I_Contact( "DB2120_MPP_ITC_IPC".RESET_FAULTS )
   END_RUNG wire#w1
   // the same network as SCL:
   #OPENED_4_ALARM := ((NOT (NOT #CYL.CLOSE_COMMAND AND NOT #CLOSE) AND #CLOSED_4_I AND #OPENED_4_I AND #CYL.SIMULTANEITY_ALARM) OR (NOT (NOT #CYL.OPEN_COMMAND AND NOT #OPEN) AND #CYL.TIME_EXCEEDED_ALARM AND NOT #OPENED_4_I) OR (#OPENED_4_ALARM AND NOT "DB2120_MPP_ITC_IPC".RESET_FAULTS)) AND #O_BYTE_0.OPENED_INPUT_4 AND "DB1401_PNEUMATIC_SYSTEM".IN_SERVICE;
END_REGION

REGION Network 34: IMMEDIATE STOP AND STOP END OF CYCLE ALARMS
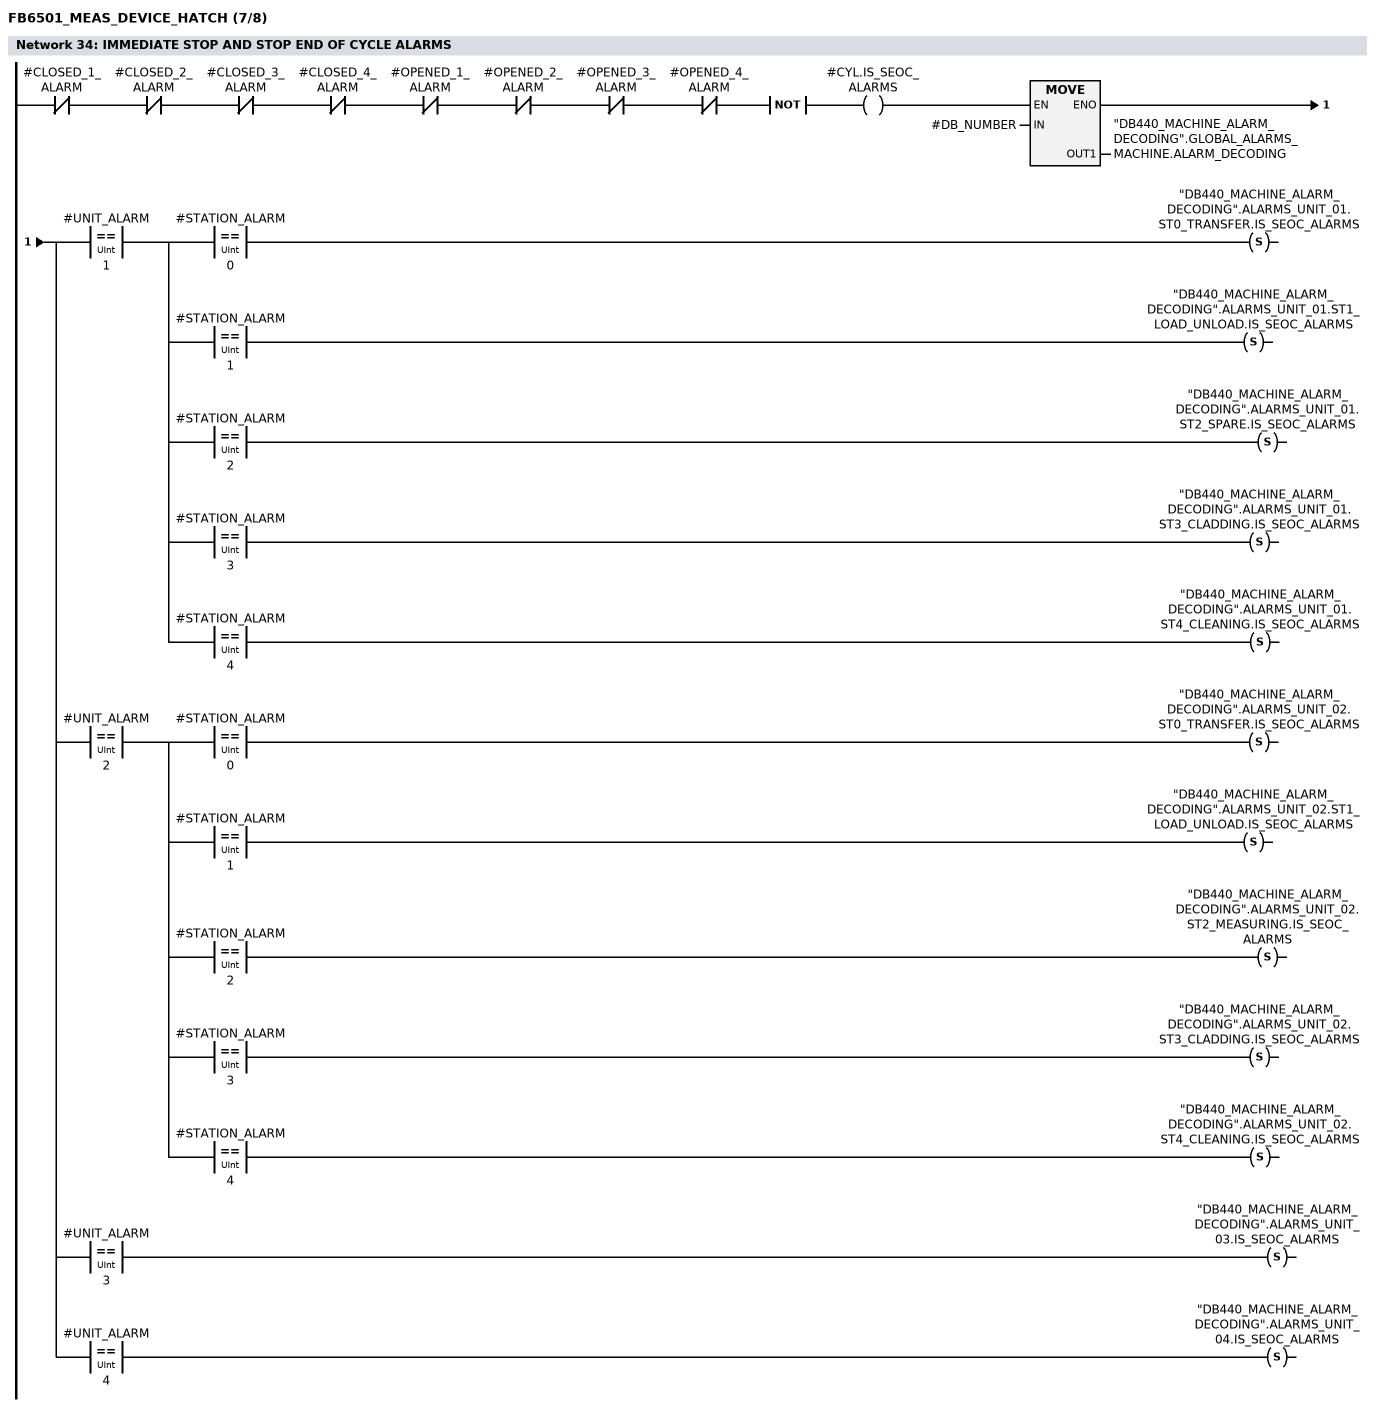
   RUNG wire#powerrail
      I_Contact( #CLOSED_1_ALARM )
      I_Contact( #CLOSED_2_ALARM )
      I_Contact( #CLOSED_3_ALARM )
      I_Contact( #CLOSED_4_ALARM )
      I_Contact( #OPENED_1_ALARM )
      I_Contact( #OPENED_2_ALARM )
      I_Contact( #OPENED_3_ALARM )
      I_Contact( #OPENED_4_ALARM )
      Not()
      Coil( #CYL.IS_SEOC_ALARMS )
      { S7_GenerateENO := "TRUE" } Move(in := #DB_NUMBER, out1 => "DB440_MACHINE_ALARM_DECODING".GLOBAL_ALARMS_MACHINE.ALARM_DECODING)
      wire#w1
      { S7_Templates := "SrcType := UInt" } EQ_Contact(in1 := #UNIT_ALARM, in2 := 1)
      wire#w2
      { S7_Templates := "SrcType := UInt" } EQ_Contact(in1 := #STATION_ALARM, in2 := 0)
      S_Coil( "DB440_MACHINE_ALARM_DECODING".ALARMS_UNIT_01.ST0_TRANSFER.IS_SEOC_ALARMS )
   END_RUNG
   RUNG wire#w2
      { S7_Templates := "SrcType := UInt" } EQ_Contact(in1 := #STATION_ALARM, in2 := 1)
      S_Coil( "DB440_MACHINE_ALARM_DECODING".ALARMS_UNIT_01.ST1_LOAD_UNLOAD.IS_SEOC_ALARMS )
   END_RUNG
   RUNG wire#w2
      { S7_Templates := "SrcType := UInt" } EQ_Contact(in1 := #STATION_ALARM, in2 := 2)
      S_Coil( "DB440_MACHINE_ALARM_DECODING".ALARMS_UNIT_01.ST2_SPARE.IS_SEOC_ALARMS )
   END_RUNG
   RUNG wire#w2
      { S7_Templates := "SrcType := UInt" } EQ_Contact(in1 := #STATION_ALARM, in2 := 3)
      S_Coil( "DB440_MACHINE_ALARM_DECODING".ALARMS_UNIT_01.ST3_CLADDING.IS_SEOC_ALARMS )
   END_RUNG
   RUNG wire#w2
      { S7_Templates := "SrcType := UInt" } EQ_Contact(in1 := #STATION_ALARM, in2 := 4)
      S_Coil( "DB440_MACHINE_ALARM_DECODING".ALARMS_UNIT_01.ST4_CLEANING.IS_SEOC_ALARMS )
   END_RUNG
   RUNG wire#w1
      { S7_Templates := "SrcType := UInt" } EQ_Contact(in1 := #UNIT_ALARM, in2 := 2)
      wire#w3
      { S7_Templates := "SrcType := UInt" } EQ_Contact(in1 := #STATION_ALARM, in2 := 0)
      S_Coil( "DB440_MACHINE_ALARM_DECODING".ALARMS_UNIT_02.ST0_TRANSFER.IS_SEOC_ALARMS )
   END_RUNG
   RUNG wire#w3
      { S7_Templates := "SrcType := UInt" } EQ_Contact(in1 := #STATION_ALARM, in2 := 1)
      S_Coil( "DB440_MACHINE_ALARM_DECODING".ALARMS_UNIT_02.ST1_LOAD_UNLOAD.IS_SEOC_ALARMS )
   END_RUNG
   RUNG wire#w3
      { S7_Templates := "SrcType := UInt" } EQ_Contact(in1 := #STATION_ALARM, in2 := 2)
      S_Coil( "DB440_MACHINE_ALARM_DECODING".ALARMS_UNIT_02.ST2_MEASURING.IS_SEOC_ALARMS )
   END_RUNG
   RUNG wire#w3
      { S7_Templates := "SrcType := UInt" } EQ_Contact(in1 := #STATION_ALARM, in2 := 3)
      S_Coil( "DB440_MACHINE_ALARM_DECODING".ALARMS_UNIT_02.ST3_CLADDING.IS_SEOC_ALARMS )
   END_RUNG
   RUNG wire#w3
      { S7_Templates := "SrcType := UInt" } EQ_Contact(in1 := #STATION_ALARM, in2 := 4)
      S_Coil( "DB440_MACHINE_ALARM_DECODING".ALARMS_UNIT_02.ST4_CLEANING.IS_SEOC_ALARMS )
   END_RUNG
   RUNG wire#w1
      { S7_Templates := "SrcType := UInt" } EQ_Contact(in1 := #UNIT_ALARM, in2 := 3)
      S_Coil( "DB440_MACHINE_ALARM_DECODING".ALARMS_UNIT_03.IS_SEOC_ALARMS )
   END_RUNG
   RUNG wire#w1
      { S7_Templates := "SrcType := UInt" } EQ_Contact(in1 := #UNIT_ALARM, in2 := 4)
      S_Coil( "DB440_MACHINE_ALARM_DECODING".ALARMS_UNIT_04.IS_SEOC_ALARMS )
   END_RUNG
   // the same network as SCL:
   // ENO of a box is taken as its EN; it also drops when the box reports an error
   #CYL.IS_SEOC_ALARMS := NOT (NOT #CLOSED_1_ALARM AND NOT #CLOSED_2_ALARM AND NOT #CLOSED_3_ALARM AND NOT #CLOSED_4_ALARM AND NOT #OPENED_1_ALARM AND NOT #OPENED_2_ALARM AND NOT #OPENED_3_ALARM AND NOT #OPENED_4_ALARM);
   IF #CYL.IS_SEOC_ALARMS THEN
       "DB440_MACHINE_ALARM_DECODING".GLOBAL_ALARMS_MACHINE.ALARM_DECODING := #DB_NUMBER;
   END_IF;
   #_w1 := #CYL.IS_SEOC_ALARMS AND (#UNIT_ALARM = 1);
   IF #_w1 AND (#STATION_ALARM = 0) THEN
       "DB440_MACHINE_ALARM_DECODING".ALARMS_UNIT_01.ST0_TRANSFER.IS_SEOC_ALARMS := TRUE;
   END_IF;
   IF #_w1 AND (#STATION_ALARM = 1) THEN
       "DB440_MACHINE_ALARM_DECODING".ALARMS_UNIT_01.ST1_LOAD_UNLOAD.IS_SEOC_ALARMS := TRUE;
   END_IF;
   IF #_w1 AND (#STATION_ALARM = 2) THEN
       "DB440_MACHINE_ALARM_DECODING".ALARMS_UNIT_01.ST2_SPARE.IS_SEOC_ALARMS := TRUE;
   END_IF;
   IF #_w1 AND (#STATION_ALARM = 3) THEN
       "DB440_MACHINE_ALARM_DECODING".ALARMS_UNIT_01.ST3_CLADDING.IS_SEOC_ALARMS := TRUE;
   END_IF;
   IF #_w1 AND (#STATION_ALARM = 4) THEN
       "DB440_MACHINE_ALARM_DECODING".ALARMS_UNIT_01.ST4_CLEANING.IS_SEOC_ALARMS := TRUE;
   END_IF;
   #_w2 := #CYL.IS_SEOC_ALARMS AND (#UNIT_ALARM = 2);
   IF #_w2 AND (#STATION_ALARM = 0) THEN
       "DB440_MACHINE_ALARM_DECODING".ALARMS_UNIT_02.ST0_TRANSFER.IS_SEOC_ALARMS := TRUE;
   END_IF;
   IF #_w2 AND (#STATION_ALARM = 1) THEN
       "DB440_MACHINE_ALARM_DECODING".ALARMS_UNIT_02.ST1_LOAD_UNLOAD.IS_SEOC_ALARMS := TRUE;
   END_IF;
   IF #_w2 AND (#STATION_ALARM = 2) THEN
       "DB440_MACHINE_ALARM_DECODING".ALARMS_UNIT_02.ST2_MEASURING.IS_SEOC_ALARMS := TRUE;
   END_IF;
   IF #_w2 AND (#STATION_ALARM = 3) THEN
       "DB440_MACHINE_ALARM_DECODING".ALARMS_UNIT_02.ST3_CLADDING.IS_SEOC_ALARMS := TRUE;
   END_IF;
   IF #_w2 AND (#STATION_ALARM = 4) THEN
       "DB440_MACHINE_ALARM_DECODING".ALARMS_UNIT_02.ST4_CLEANING.IS_SEOC_ALARMS := TRUE;
   END_IF;
   IF #CYL.IS_SEOC_ALARMS AND (#UNIT_ALARM = 3) THEN
       "DB440_MACHINE_ALARM_DECODING".ALARMS_UNIT_03.IS_SEOC_ALARMS := TRUE;
   END_IF;
   IF #CYL.IS_SEOC_ALARMS AND (#UNIT_ALARM = 4) THEN
       "DB440_MACHINE_ALARM_DECODING".ALARMS_UNIT_04.IS_SEOC_ALARMS := TRUE;
   END_IF;
END_REGION

REGION Network 35: ANY ACTIVE ALARM
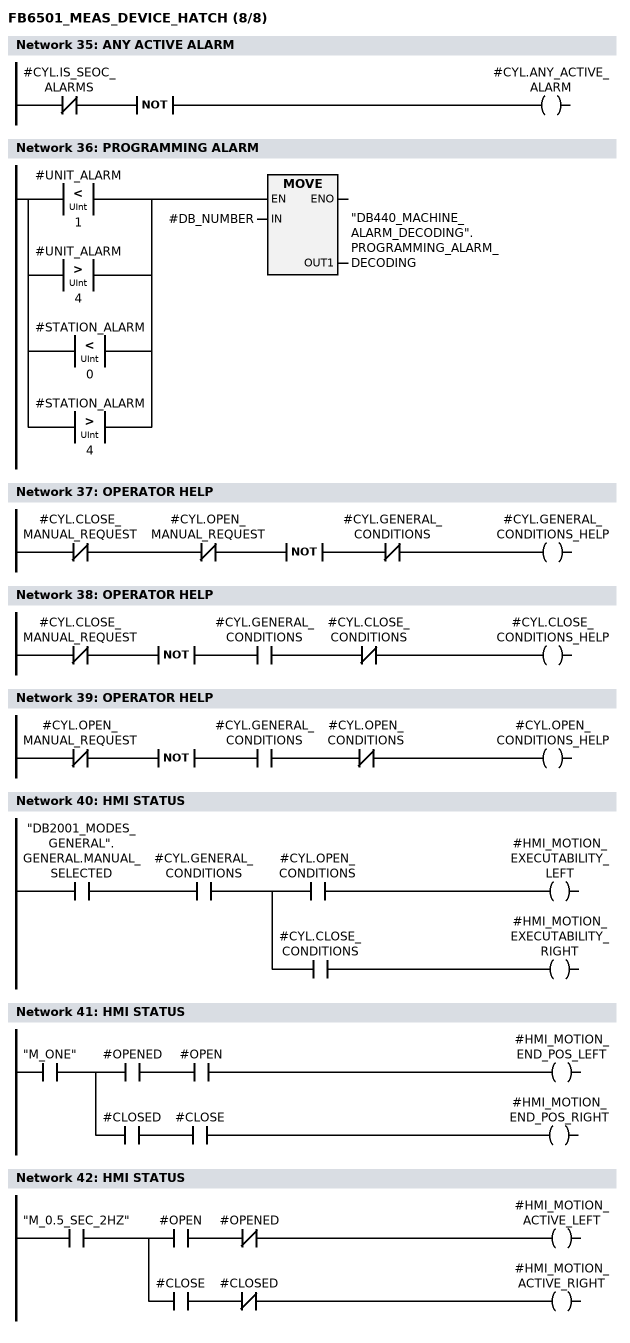
   RUNG wire#powerrail
      I_Contact( #CYL.IS_SEOC_ALARMS )
      Not()
      Coil( #CYL.ANY_ACTIVE_ALARM )
   END_RUNG
   // the same network as SCL:
   #CYL.ANY_ACTIVE_ALARM := NOT (NOT #CYL.IS_SEOC_ALARMS);
END_REGION

REGION Network 36: PROGRAMMING ALARM
   RUNG wire#powerrail
      { S7_Templates := "SrcType := UInt" } LT_Contact(in1 := #UNIT_ALARM, in2 := 1)
      wire#w1
      Move(in := #DB_NUMBER, out1 => "DB440_MACHINE_ALARM_DECODING".PROGRAMMING_ALARM_DECODING)
   END_RUNG
   RUNG wire#powerrail
      { S7_Templates := "SrcType := UInt" } GT_Contact(in1 := #UNIT_ALARM, in2 := 4)
   END_RUNG wire#w1
   RUNG wire#powerrail
      { S7_Templates := "SrcType := UInt" } LT_Contact(in1 := #STATION_ALARM, in2 := 0)
   END_RUNG wire#w1
   RUNG wire#powerrail
      { S7_Templates := "SrcType := UInt" } GT_Contact(in1 := #STATION_ALARM, in2 := 4)
   END_RUNG wire#w1
   // the same network as SCL:
   IF (#UNIT_ALARM < 1) OR (#UNIT_ALARM > 4) OR (#STATION_ALARM < 0) OR (#STATION_ALARM > 4) THEN
       "DB440_MACHINE_ALARM_DECODING".PROGRAMMING_ALARM_DECODING := #DB_NUMBER;
   END_IF;
END_REGION

REGION Network 37: OPERATOR HELP
   RUNG wire#powerrail
      I_Contact( #CYL.CLOSE_MANUAL_REQUEST )
      I_Contact( #CYL.OPEN_MANUAL_REQUEST )
      Not()
      I_Contact( #CYL.GENERAL_CONDITIONS )
      Coil( #CYL.GENERAL_CONDITIONS_HELP )
   END_RUNG
   // the same network as SCL:
   #CYL.GENERAL_CONDITIONS_HELP := NOT (NOT #CYL.CLOSE_MANUAL_REQUEST AND NOT #CYL.OPEN_MANUAL_REQUEST) AND NOT #CYL.GENERAL_CONDITIONS;
END_REGION

REGION Network 38: OPERATOR HELP
   RUNG wire#powerrail
      I_Contact( #CYL.CLOSE_MANUAL_REQUEST )
      Not()
      Contact( #CYL.GENERAL_CONDITIONS )
      I_Contact( #CYL.CLOSE_CONDITIONS )
      Coil( #CYL.CLOSE_CONDITIONS_HELP )
   END_RUNG
   // the same network as SCL:
   #CYL.CLOSE_CONDITIONS_HELP := NOT (NOT #CYL.CLOSE_MANUAL_REQUEST) AND #CYL.GENERAL_CONDITIONS AND NOT #CYL.CLOSE_CONDITIONS;
END_REGION

REGION Network 39: OPERATOR HELP
   RUNG wire#powerrail
      I_Contact( #CYL.OPEN_MANUAL_REQUEST )
      Not()
      Contact( #CYL.GENERAL_CONDITIONS )
      I_Contact( #CYL.OPEN_CONDITIONS )
      Coil( #CYL.OPEN_CONDITIONS_HELP )
   END_RUNG
   // the same network as SCL:
   #CYL.OPEN_CONDITIONS_HELP := NOT (NOT #CYL.OPEN_MANUAL_REQUEST) AND #CYL.GENERAL_CONDITIONS AND NOT #CYL.OPEN_CONDITIONS;
END_REGION

REGION Network 40: HMI STATUS
   RUNG wire#powerrail
      Contact( "DB2001_MODES_GENERAL".GENERAL.MANUAL_SELECTED )
      Contact( #CYL.GENERAL_CONDITIONS )
      wire#w1
      Contact( #CYL.OPEN_CONDITIONS )
      Coil( #HMI_MOTION_EXECUTABILITY_LEFT )
   END_RUNG
   RUNG wire#w1
      Contact( #CYL.CLOSE_CONDITIONS )
      Coil( #HMI_MOTION_EXECUTABILITY_RIGHT )
   END_RUNG
   // the same network as SCL:
   #_w1 := "DB2001_MODES_GENERAL".GENERAL.MANUAL_SELECTED AND #CYL.GENERAL_CONDITIONS;
   #HMI_MOTION_EXECUTABILITY_LEFT := #_w1 AND #CYL.OPEN_CONDITIONS;
   #HMI_MOTION_EXECUTABILITY_RIGHT := #_w1 AND #CYL.CLOSE_CONDITIONS;
END_REGION

REGION Network 41: HMI STATUS
   RUNG wire#powerrail
      Contact( "M_ONE" )
      wire#w1
      Contact( #OPENED )
      Contact( #OPEN )
      Coil( #HMI_MOTION_END_POS_LEFT )
   END_RUNG
   RUNG wire#w1
      Contact( #CLOSED )
      Contact( #CLOSE )
      Coil( #HMI_MOTION_END_POS_RIGHT )
   END_RUNG
   // the same network as SCL:
   #HMI_MOTION_END_POS_LEFT := "M_ONE" AND #OPENED AND #OPEN;
   #HMI_MOTION_END_POS_RIGHT := "M_ONE" AND #CLOSED AND #CLOSE;
END_REGION

REGION Network 42: HMI STATUS
   RUNG wire#powerrail
      Contact( "M_0.5_SEC_2HZ" )
      wire#w1
      Contact( #OPEN )
      I_Contact( #OPENED )
      Coil( #HMI_MOTION_ACTIVE_LEFT )
   END_RUNG
   RUNG wire#w1
      Contact( #CLOSE )
      I_Contact( #CLOSED )
      Coil( #HMI_MOTION_ACTIVE_RIGHT )
   END_RUNG
   // the same network as SCL:
   #HMI_MOTION_ACTIVE_LEFT := "M_0.5_SEC_2HZ" AND #OPEN AND NOT #OPENED;
   #HMI_MOTION_ACTIVE_RIGHT := "M_0.5_SEC_2HZ" AND #CLOSE AND NOT #CLOSED;
END_REGION
END_FUNCTION_BLOCK
